// TIA Portal V17 export
// export: Created 2023-04-07T07:34:43.6013741Z, ExportSetting WithDefaults, DisplayName Totally Integrated Automation Portal, DisplayVersion V17 Update 4, DisplayName TIA Portal Openness, DisplayVersion V17 Update 4, DisplayName TIA Portal Version Control Interface, DisplayVersion V17, DisplayName STEP 7 Professional, DisplayVersion V17 Update 4, DisplayName STEP 7 Safety, DisplayVersion V17, DisplayName WinCC Professional, DisplayVersion V17 Update 4
FUNCTION "PCS W (S)_2" : Void   // FC52, LAD
TITLE = ModBus TCP for PCS Power Electronics
{ S7_Optimized_Access := 'TRUE' }
VERSION : 0.1
// stored: AutoNumber true, IsIECCheckEnabled false, SetENOAutomatically false, UDAEnableTagReadback false
   VAR_TEMP
      rSS1PacRef : Real;
      rSS2PacRef : Real;
      rSS1QacRef : Real;
      rSS2QacRef : Real;
      rSnHalfPE : Real;
      rQacRef : Real;
      uiQacRef : UInt;
   END_VAR
BEGIN
END_FUNCTION
